Staubli VAL3: getTraj.pgx

public program getTraj(Trajectory& x_tTrajectory (dimensions=1))
  local num l_nSize
begin
  // mutex it
  setMutex(bActionMutex)
  // get the first Traj
  x_tTrajectory=tTrajCycle[0]
  // release
  bActionMutex=false
end
